{attribute 'qualified_only'}
{attribute 'strict'}
{attribute 'to_string'}
TYPE MotorZuignaptoestand :
(
	Lang := 0,
	Kort,
	Ingaand,
	Uitgaand,
	error
);
END_TYPE

(* stored: Version 1.1.0.1
   DUT MotorZuignaptoestand: Id {4d80b3bd-69fb-4710-a150-94b22ebdfa7f} *)
